// TIA Portal V21 export
FUNCTION_BLOCK "__PI_CREATEFB_NAME__"   // FB__PI_CREATEFB_NUMBER__, SCL
{ S7_Optimized_Access := 'TRUE' }
// Minimal disposable SCL FB template imported by TiaLocalBridge.
// stored: IsIECCheckEnabled true, MemoryReserve 100, SetENOAutomatically true
BEGIN
   REGION Generated template
     //Minimal FB template created by TiaLocalBridge.
   END_REGION Generated template
END_FUNCTION_BLOCK
